{attribute 'reflection'}
FUNCTION_BLOCK FB_PitchControl_old
VAR_IN_OUT
	Pitch : HOMS_PitchMechanism;
END_VAR
VAR_INPUT
	ManualMode	:	BOOL := FALSE;
END_VAR
VAR_OUTPUT
	q_xError	:	BOOL;
	q_xDone	:	BOOL;
END_VAR
VAR
	//Introspection
	//////////////////////////////
		{attribute 'instance-path'}
		{attribute 'no_init'}
		POUName	:	STRING; //Name of the POU for logging/error reporting
	
	
	//FB Boilerplate
	//////////////////////
		stDiag	:	ST_fbDiagnostics;
		fbFormatString	:	FB_FormatString;
		
	
	PC_State : E_PitchControl := PCM_Init;
	
	PiezoRelMax: LREAL; //High side of piezo range
	cPiezoMax: LREAL; //Nominal range of the piezo
	aM1PiezoCal: LREAL; //Placeholder for piezo calibration table
	PiezoRelMin: LREAL; //Low side of piezo range
	PiezoPosition: LREAL; //Estimated piezo extension
	// um, set based on piezo actuator extension
	cPiezo50Perc	: 	REAL := 45; //um
	cPiezo50PercTol	:	REAL := 1; //um
	

	// Previously requested position. Set at the end of a move.
	PreviousReqAbsPos: LREAL;
	// Original position requested, before soft limits
	OriginalPosRequest: LREAL;
	
	//Axis Control Blocks
	/////////////////////////////
		//fbStepper	:	FB_BasicAxisControl;
		fbPiezoControl	:	FB_PiezoControl; //Closed-loop fine-pitch adjustment.
		mcStepperPower: MC_Power;
		mcStepperReset: MC_Reset;
		mcStepperMovAbs: MC_MoveAbsolute;
	
	
	//Triggers
	//////////////////////////////
		rtStartMove	:	R_TRIG;
		rtReset:	R_TRIG;
		rtEnable:	R_TRIG;
		rtManualMode:	R_TRIG;
		ftManualMode	:	F_TRIG;
	// Request for voltage mode from the coarse 50% move step.
	Coarse50VoltageMode: BOOL := FALSE;
	// Coarse 50% piezo move start request
	Coarse50PiezoMove: BOOL := FALSE;
END_VAR

(* HOMS Pitch Control
A. Wallace

The HOMS Pitch mechanism consists of a stepper and piezo that work together to adjust
the pitch of the mirror assembly.

Pitch control state machine

If the target position is beyond the range of the piezo mechanism,
execute a coarse pitch move with the stepper. 
The target of the coarse move shall be set to the requested position. 
Once coarse motion has completed the coarse motion drive position 
correction output shall be set to zero.

Fine pitch motion with the piezo will be initiated to finish closing the loop.

The piezo mechanism can actuate ~ 180urad or 90um.

*)

rtStartMove(CLK:=Pitch.Axis.xStartAbsMove);
rtReset(CLK:=Pitch.Axis.xReset);
rtEnable(CLK:=Pitch.Axis.xEnable);

//Manual mode switching logic
/////////////////////////////////////
	rtManualMode(CLK:=ManualMode);
	ftManualMode(CLK:=ManualMode);
	A_ModeSwitch();



(* In expert mode we want individual control of both the piezo and stepper.
We still want the piezo and stepper to respect the limit switches, and 
soft limits if possible.
*)

//State Machine
//////////////////////////////////
CASE PC_State OF
	PCM_Init: 
		//Initialize stepper motor mc power block
		mcStepperPower.Enable S= rtEnable.Q;
		IF mcStepperPower.Status THEN
			PC_State := PCM_Standby;
		ELSIF mcStepperPower.Error THEN
			PC_State := PCM_StepperError;
			// <TODO> error message
		END_IF
	PCM_Standby:
		//We should only listen for move attempts if the interlock is good.
		IF Pitch.Axis.i_xMotorInterlock THEN
			IF rtStartMove.Q THEN
				IF (PreviousReqAbsPos <> Pitch.Axis.rReqAbsPos) THEN
					//We don't want to initiate any kind of a move if we don't have to.
					IF 	Pitch.Axis.rReqAbsPos > Pitch.ReqPosLimHi OR Pitch.Axis.rReqAbsPos < Pitch.ReqPosLimLo THEN
						//Requested move is outside of travel limits
						OriginalPosRequest	:= Pitch.Axis.rReqAbsPos;
						Pitch.Axis.rReqAbsPos := LIMIT(Pitch.ReqPosLimLo, Pitch.Axis.rReqAbsPos, Pitch.ReqPosLimHi);
						//Only want to log one warning about a bad position request.
						IF OriginalPosRequest <> Pitch.Axis.rReqAbsPos THEN
							//Log a warning
							fbFormatString.sFormat := 'Pitch position requested outside of range fb (%s), reset within limits %d';
							fbFormatString.arg1 := F_STRING(POUName);
							fbFormatString.arg2 := F_LREAL(OriginalPosRequest);
							fbFormatString(sOut=>fbLogMessage.i_sMsg);
							fbLogMessage(i_eSevr:= Warning, i_eSubsystem:=gDefaultSubsystem);
						END_IF
					END_IF
					
					q_xDone := FALSE;
					PC_State := PCM_MoveRequested;
				END_IF
			END_IF
		ELSIF rtStartMove.Q AND NOT Pitch.Axis.i_xMotorInterlock THEN
			Pitch.Axis.xStartAbsMove := FALSE;
			//<TODO> Maybe we implement a log here when logging levels can be adjusted
		ELSE
			Pitch.Axis.xStartAbsMove := FALSE;
		END_IF
			
	PCM_MoveRequested: 
		//A move has been requested, is it within range of the piezo?
		PiezoPosition := F_PiezoPosition(rPiezoVoltage := Pitch.Piezo.rActVoltage, aM1PiezoCal);
		PiezoRelMax := Pitch.Stepper.stAxis.NcToPlc.ActPos + 
			cPiezoMax - PiezoPosition;
		PiezoRelMin := Pitch.Stepper.stAxis.NcToPlc.ActPos - PiezoPosition;
		IF Pitch.Axis.rReqAbsPos > PiezoRelMax OR Pitch.Axis.rReqAbsPos < PiezoRelMin THEN
			// Out of range, head to coarse move
			PC_State := PCM_Coarse50Piezo;
		ELSE
			//Move is within the nominal range of the piezo
			PC_State := PCM_FineMove;
		END_IF
	PCM_Coarse50Piezo:
		//A coarse move uses the stepper to do a best-effort position
		//First set the piezo to nominal 50% extension using absolute position request
		//////////////////////////////////////////////////////////////////////////////
			//PiezoPosition := F_PiezoPosition(rPiezoVoltage := Pitch.Piezo.rActVoltage, aM1PiezoCal);
			//Pitch.Piezo.rReqAbsPos := cPiezo50Perc;
			
		//Alternatively, set the piezo voltage to ~50% manually using voltage mode
		/////////////////////////////////////////////////////////
			//Coarse50VoltageMode	:= TRUE;
			//Coarse50VoltageMode R= fbPiezoControl.xDone OR fbPiezoControl.xError;
			
		Coarse50PiezoMove := TRUE;
		Coarse50PiezoMove R= fbPiezoControl.xDone OR fbPiezoControl.xError;
		IF fbPiezoControl.xDone THEN
			//Piezo has moved to 50% position, finish with the stepper
			PC_State := PCM_CoarseMove;
			Pitch.Piezo.xStartAbsMove := FALSE;
		ELSIF fbPiezoControl.xError THEN
			//Piezo move timed out, something is wrong
			fbFormatString.sFormat := 'Piezo move to 50% encountered an error in %s';
			fbFormatString.arg1 := F_STRING(POUName);
			fbFormatString(sOut=>fbLogMessage.i_sMsg);
			fbLogMessage(i_eSevr:= Critical, i_eSubsystem:=gDefaultSubsystem);
			PC_State := PCM_PiezoError;
		END_IF
	PCM_CoarseMove: 
		//With the piezo at a nom 50% extension, move the stepper to requested position
		mcStepperMovAbs.Position := Pitch.Axis.rReqAbsPos;
		mcStepperMovAbs.Execute := TRUE;
		mcStepperMovAbs.Execute R= mcStepperMovAbs.Busy OR mcStepperMovAbs.Error;
		//If the coarse move is complete, finish position correction with the piezo
		IF mcStepperMovAbs.Done THEN
			PC_State := PCM_FineMove;
		ELSIF mcStepperMovAbs.Error THEN
			PC_State := PCM_StepperError;
			//Stepper fb has encountered an error, pass a message to the logger
			fbFormatString.sFormat := 'Pitch coarse stepper move encountered an error in: %s, error id %d';
			fbFormatString.arg1 := F_STRING(POUName);
			fbFormatString.arg2 := F_UDINT(mcStepperMovAbs.ErrorID);
			fbFormatString(sOut=>fbLogMessage.i_sMsg);
			fbLogMessage(i_eSevr:= Critical, i_eSubsystem:=gDefaultSubsystem);
		END_IF
	PCM_FineMove:	
		fbPiezoControl.xExecute := TRUE;
		fbPiezoControl.xExecute R= fbPiezoControl.xBusy OR fbPiezoControl.xError;
		Pitch.Piezo.rReqAbsPos := Pitch.Axis.rReqAbsPos;
		//If the piezo move is complete, this move is done.
		IF fbPiezoControl.xDone THEN
			PC_State := PCM_Done;
		ELSIF fbPiezoControl.xError THEN
			PC_State := PCM_PiezoError;
			fbFormatString.sFormat := 'Pitch fine move encountered an error in: %s';
			fbFormatString.arg1 := F_STRING(POUName);
			fbFormatString(sOut=>fbLogMessage.i_sMsg);
		END_IF
	PCM_Done:
		//Set the previously requested position here
		PreviousReqAbsPos := Pitch.Axis.rReqAbsPos;
		//Indicate we're done
		q_xDone	:= TRUE;
		//Move back to standby
		PC_State := PCM_Standby;
	PCM_StepperError:
		IF mcStepperReset.Done THEN
			PC_State := PCM_Init; 
		END_IF
	PCM_PiezoError:
		IF rtReset.Q THEN
			PC_State := PCM_Init;
		END_IF
	PCM_OtherError:
		IF rtReset.Q THEN
			PC_State := PCM_Init;
		END_IF
	
END_CASE

//Simple test to determine if we have an error or not.
q_xError := PC_State >= PCM_Error;



A_MotionFB();

ACTION A_ModeSwitch:
(* When switching between modes, we need to make sure all the executes/ mode switches, etc. are cleared *)

// Automatic to manual
/////////////////////////////
IF rtManualMode.Q THEN
	Coarse50VoltageMode := FALSE;
	mcStepperPower.Enable := FALSE;
	mcStepperMovAbs.Execute := FALSE;
	fbPiezoControl.xExecute := FALSE;
END_IF

// Manual to automatic
//////////////////////////////
IF ftManualMode.Q THEN
	;
END_IF
END_ACTION

ACTION A_MotionFB:
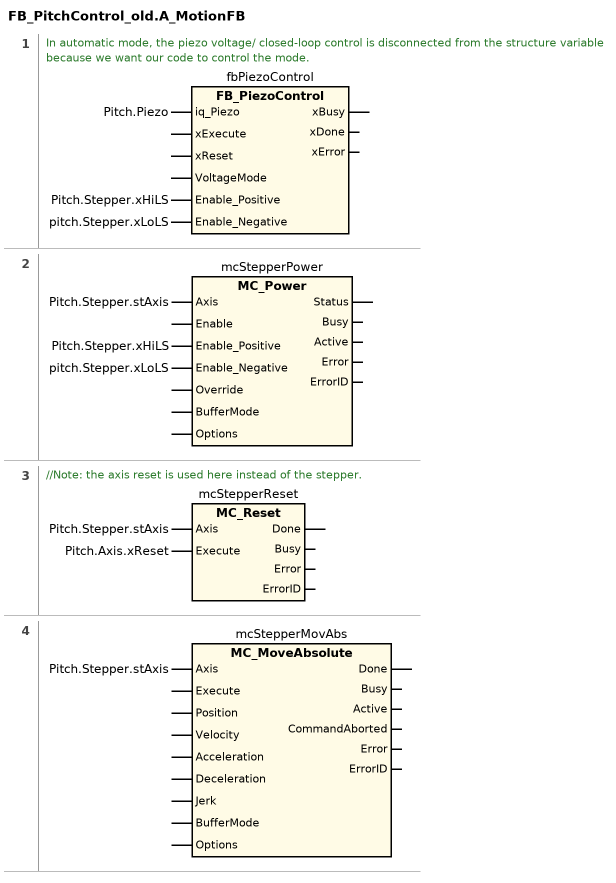
// NETWORK 1
// In automatic mode, the piezo voltage/ closed-loop control is disconnected from the structure variable
// because we want our code to control the mode.
fbPiezoControl(
    iq_Piezo := Pitch.Piezo,
    Enable_Positive := Pitch.Stepper.xHiLS,
    Enable_Negative := pitch.Stepper.xLoLS); // FB_PiezoControl

// NETWORK 2
mcStepperPower(
    Axis := Pitch.Stepper.stAxis,
    Enable_Positive := Pitch.Stepper.xHiLS,
    Enable_Negative := pitch.Stepper.xLoLS); // MC_Power

// NETWORK 3
// //Note: the axis reset is used here instead of the stepper.
mcStepperReset(Axis := Pitch.Stepper.stAxis, Execute := Pitch.Axis.xReset); // MC_Reset

// NETWORK 4
mcStepperMovAbs(Axis := Pitch.Stepper.stAxis); // MC_MoveAbsolute
END_ACTION

END_FUNCTION_BLOCK

(* stored: Version 1.1.0.1, ProductVersion 3.1.4020.12
   POU FB_PitchControl_old: Id {5d7f0ff1-cf67-4bce-80fc-4e4ac0fd9e20}, SpecialFunc None
   Action A_ModeSwitch: Id {aab9346d-393d-4f86-a5e3-e32335e00aef}
   Action A_MotionFB: Id {9e229e50-6d9e-468a-a7d2-47fa9301fb05} *)
